// TIA Portal V20 export
TYPE "LER_typeCommunicationData_I2S"
// stored: Access Published
   STRUCT
      UnitStatus : "LER_typeCommunicationUnitStatus";
      UnitHmiData : Array[1..50] of "LER_typeUnitHmiData";
      InterfaceData : "LER_typeCommunicationInterfaceData";
   END_STRUCT;
   // // InterfaceData."Bool"[0] : Heartbeat
   // // InterfaceData."Bool"[1] : ReadyForOperation
   // // InterfaceData."Bool"[2] : ReachedHome
   // // InterfaceData."Bool"[3] : MachineInOperation
   // // InterfaceData."Bool"[4] : LoaderOutsideModule
   // // InterfaceData."Bool"[5] : LoaderOutsideCollision
   // // InterfaceData."Bool"[10] : PartClamped
   // // InterfaceData."Bool"[11] : PartUnclamped
   // // InterfaceData."Bool"[16] : RequestUnclamp
   // // InterfaceData."Bool"[17] : PartOn
   // // InterfaceData."Bool"[18] : RequestPart
   // // InterfaceData."Bool"[19] : OnPositionUnloading
   // // InterfaceData."Bool"[22] : RequestCollisionON
   // // InterfaceData."Bool"[23] : UnoadComplete
   // // InterfaceData."Bool"[26] : DataCatchUp
   // // InterfaceData."Bool"[27] : DataCompareOK
   // // InterfaceData."Bool"[28] : DataDeleted
   // // InterfaceData."Bool"[32] : NG RequestPart
   // // InterfaceData."Bool"[33] : NG RequestUnclamp
   // // InterfaceData."Bool"[34] : NG UnoadComplete
   // // InterfaceData."Bool"[40] : HoursTestMode.On/Off.Status
   // // InterfaceData."Bool"[41] : HourTestMode_Completed
   // // InterfaceData."Bool"[42] : CapabilityMode.On/Off.Status
   // // InterfaceData."Bool"[43] : CapabilityMode_Completed
   // // InterfaceData."Bool"[48] : ReturnToHome
   // // InterfaceData."Bool"[49] : AutoStart
   // // InterfaceData."Bool"[50] : EndOfCycle
   // // InterfaceData."Bool"[51] : RequestGateOpen
   // // InterfaceData.LReal[0] : HoursTestMode_SetTime
   // // InterfaceData.LReal[1] : HoursTestMode_TimeLeft
   // // InterfaceData.LReal[2] : Capability CurrentCount
   // // InterfaceData.LReal[3] : CapabilityCountSetValue
END_TYPE
